(* PLC project test.project, CODESYS CODESYS V3.5 SP18 Patch 3 *)
(* stored: creationDateTime 2023-02-15T12:59:17.1674637, modificationDateTime 2023-02-15T12:50:55.5586453 *)

PROGRAM PLC_PRG
  VAR
    trans0 : BOOL;
    trans1 : BOOL;
    trans2 : BOOL;
    trans4 : BOOL;
    trans5 : BOOL;
    trans6 : BOOL;
    trans7 : BOOL;
    trans8 : BOOL;
    trans9 : BOOL;
    trans10 : BOOL := 0;
    out0 : BOOL;
    trans12 : BOOL;
    trans13 : BOOL;
    trans11 : BOOL;
    trans15 : BOOL;
    trans14 : BOOL;
    trans16 : BOOL;
    trans17 : BOOL;
    out2 : BOOL;
    T1 : TIME := TIME#360m0s0ms;
    T2 : TIME := TIME#4ms;
    out1 : BOOL;
  END_VAR

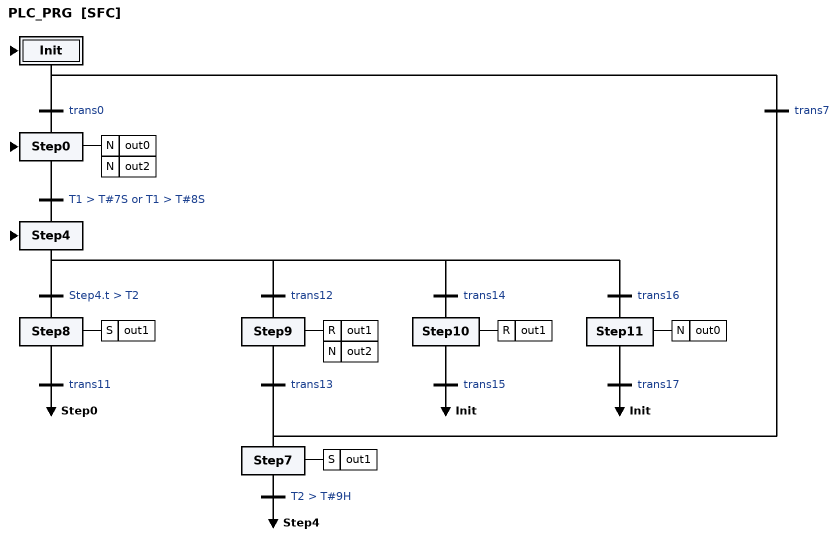
INITIAL_STEP Init:
END_STEP
TRANSITION FROM Init TO Step0
  := trans0;
END_TRANSITION
TRANSITION FROM Init TO Step7
  := trans7;
END_TRANSITION
STEP Step0:
  out0(N);
  out2(N);
END_STEP
TRANSITION FROM Step0 TO Step4
  := T1 > T#7S or T1 > T#8S;
END_TRANSITION
STEP Step7:
  out1(S);
END_STEP
TRANSITION FROM Step7 TO Step4
  := T2 > T#9H;
END_TRANSITION
STEP Step4:
END_STEP
TRANSITION FROM Step4 TO Step8
  := Step4.t > T2;
END_TRANSITION
TRANSITION FROM Step4 TO Step9
  := trans12;
END_TRANSITION
TRANSITION FROM Step4 TO Step10
  := trans14;
END_TRANSITION
TRANSITION FROM Step4 TO Step11
  := trans16;
END_TRANSITION
STEP Step8:
  out1(S);
END_STEP
TRANSITION FROM Step8 TO Step0
  := trans11;
END_TRANSITION
STEP Step9:
  out1(R);
  out2(N);
END_STEP
TRANSITION FROM Step9 TO Step7
  := trans13;
END_TRANSITION
STEP Step10:
  out1(R);
END_STEP
TRANSITION FROM Step10 TO Init
  := trans15;
END_TRANSITION
STEP Step11:
  out0(N);
END_STEP
TRANSITION FROM Step11 TO Init
  := trans17;
END_TRANSITION
END_PROGRAM
